// Mitsubishi GX Works2 project: MPS 장비 제어하기 2-1   PLC: Q03UDV

PROGRAM MAIN
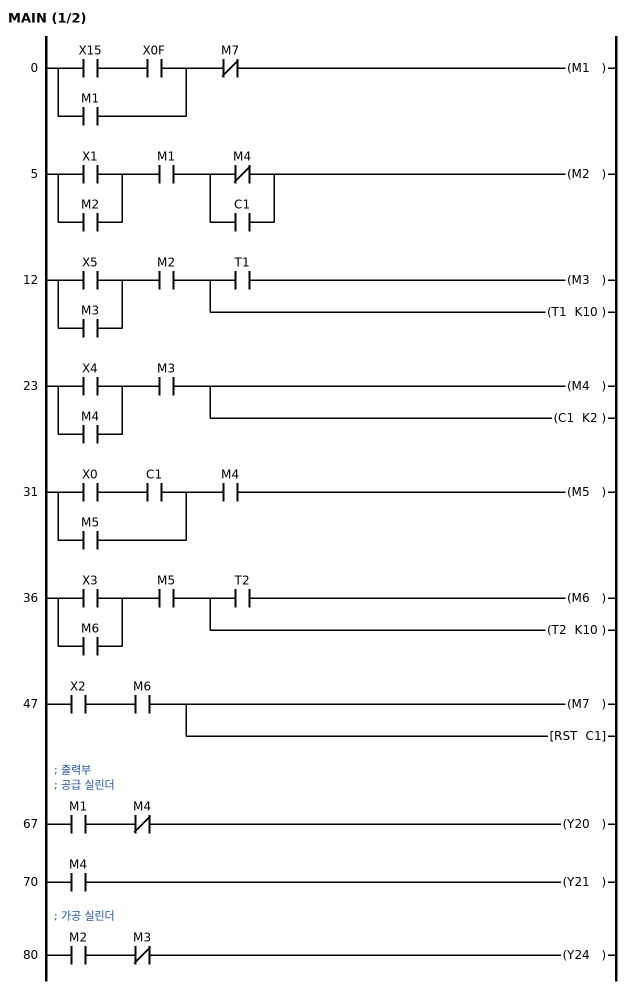
0     LD      X15
      AND     X0F
      OR      M1
      ANI     M7
      OUT     M1
5     LD      X1
      OR      M2
      AND     M1
      LDI     M4
      OR      C1
      ANB
      OUT     M2
12    LD      X5
      OR      M3
      AND     M2
      MPS
      AND     T1
      OUT     M3
      MPP
      OUT     T1 K10
23    LD      X4
      OR      M4
      AND     M3
      OUT     M4
      OUT     C1 K2
31    LD      X0
      AND     C1
      OR      M5
      AND     M4
      OUT     M5
36    LD      X3
      OR      M6
      AND     M5
      MPS
      AND     T2
      OUT     M6
      MPP
      OUT     T2 K10
47    LD      X2
      AND     M6
      OUT     M7
      RST     C1
; 출력부
; 공급 실린더
67    LD      M1
      ANI     M4
      OUT     Y20
70    LD      M4
      OUT     Y21
; 가공 실린더
80    LD      M2
      ANI     M3
      OUT     Y24
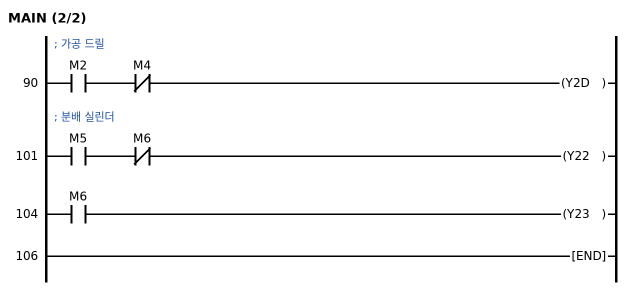
; 가공 드릴
90    LD      M2
      ANI     M4
      OUT     Y2D
; 분배 실린더
101   LD      M5
      ANI     M6
      OUT     Y22
104   LD      M6
      OUT     Y23
106   END
END_PROGRAM
